Yaskawa INFORM job: _DEL22.JBI

/JOB
//NAME _DEL22
//POS
///NPOS 0,0,0,0,0,0
//INST
///DATE 2018/08/30 09:57
///ATTR SC,RW,SY
///LVARS 5,0,5,0,0,0,0,0
NOP
END
